// P1 - STRUCT - 
// Rev 1.0 - Sepember 6, 2024

TYPE Blank : 
	STRUCT
		cooling_pump : BYTE;
		dead_air_pump : BYTE;
		steam_system : BYTE;
		purge_assist : BYTE;
		test : BYTE;
	END_STRUCT
END_TYPE

(* stored: Version 1.1.0.1, ProductVersion 3.1.4024.13
   DUT Blank: Id {d9fafee2-97c9-4451-ad9d-ad3a6c3d8935} *)
